// TwinCAT 3 PLC project TAC_Events
// Title: TAC_Events
// Company: Timberline Automation and Control Co.
// Author: Mit Patel
// ProjectVersion: 0.1.1.2
// Description: V0.1.1.0 - Initial V0.1.1.1 - Create RPC Sink V0.1.1.2 - Separate Buffer and Sink Interfaces
// ProgramVersion: 3.1.4026.19
// libraries:
//   Tc2_EtherCAT, * (Beckhoff Automation GmbH)
//   Tc2_Standard, * (Beckhoff Automation GmbH)
//   Tc2_System, * (Beckhoff Automation GmbH)
//   Tc2_Utilities, * (Beckhoff Automation GmbH)
//   Tc3_JsonXml, * (Beckhoff Automation GmbH)
// project tree:
//   ImportUtilities/ LogConfig.TcGVL
//   ImportUtilities/Logger/ E_LogSeverity.TcDUT, FB_LogErrorEdge.TcPOU, FB_LogInfoEdge.TcPOU, FB_LogOnEdge.TcPOU, FB_LogWarningEdge.TcPOU, F_LogDebug.TcPOU, F_LogError.TcPOU, F_Logger.TcPOU, F_LogInfo.TcPOU, F_LogWarning.TcPOU, I_ExternalLogger.TcIO
//   ImportUtilities/String/ F_Concat3.TcPOU, F_Concat4.TcPOU, F_Concat5.TcPOU, F_Concat6.TcPOU, F_Concat7.TcPOU, F_StringToTarg.TcPOU, F_TargToString.TcPOU, LongString.TcDUT
//   ImportUtilities/String/Large Concats/ F_ClearLarge.TcPOU, F_Concat3_Large.TcPOU, F_Concat4_Large.TcPOU, F_Concat5_Large.TcPOU, F_Concat6_Large.TcPOU, F_Concat7_Large.TcPOU, F_ConcatLarge.TcPOU
//   Library/EventLogger/EventBuffers/ T_JsonEventBuffer.TcPOU
//   Library/EventLogger/EventSinks/ T_RpcEventSink.TcPOU (not stored), FB_CsvFileEventSink.TcPOU (not stored)
//   Library/EventLogger/Interfaces/ I_EventSink.TcIO (not stored), I_EventBuffer.TcIO (not stored), I_EventLogger.TcIO (not stored), I_Logger.TcIO, I_EventSeverityHandler.TcIO (not stored), I_EventSinkHandler.TcIO
//   Library/Structs/ ST_EventMessageBuffer.TcDUT (not stored), ST_EventMessageBufferPool.TcDUT, ST_EventMessageParams.TcDUT, T_BufferString.TcDUT, T_MessageString.TcDUT (not stored)
//   Library/EventLogger/Bases/ T_InstanceNameBase.TcPOU (not stored)
//   Library/EventLogger/Functions/ F_GetLogSeverityFromTcEventSeverity.TcPOU (not stored)
//   Library/EventLogger/ T_EventLogger.TcPOU (not stored), T_Logger.TcPOU
//   Library/GVLs/ Events.TcGVL, EventsConfig.TcGVL (not stored)
//   Library/Time/ FB_UnixTimestamp.TcPOU, I_TimeProvider.TcIO (not stored)
//   Project Information/ F_GetCompany.TcPOU, F_GetTitle.TcPOU, F_GetVersion.TcPOU (not stored)
//   Version/ Global_Version.TcGVL
// real-time tasks:
//   TASK PlcTask: cycle T#10ms, priority 20, ADS port 350
//   TASK PlcTask1: cycle T#10ms, priority 21, ADS port 351

// ---- ImportUtilities/Logger/E_LogSeverity.TcDUT
{attribute 'qualified_only'}
TYPE
   E_LogSeverity :
   (
      Debug := 0,
      Info := ADSLOG_MSGTYPE_HINT,
      Warning := ADSLOG_MSGTYPE_WARN,
      Error := ADSLOG_MSGTYPE_ERROR,
      None := 1000
   ) DWORD;
END_TYPE

// ---- ImportUtilities/String/LongString.TcDUT
TYPE
   LongString : STRING(StringsParams.MAX_STRING_LENGTH);
END_TYPE // use StringsParams.MAX_STRING_LENGTH to adjust length

// ---- Library/Structs/ST_EventMessageBufferPool.TcDUT
{attribute 'pack_mode' := '0'}
TYPE ST_EventMessageBufferPool :
STRUCT
  bufferCount : UINT := EventsConfig.MAX_BUFFERS;
	currentDataBufferIndex : UINT := 0;
	dataBuffers : ARRAY [1..EventsConfig.MAX_BUFFERS] OF ST_EventMessageBuffer;
END_STRUCT
END_TYPE

// ---- Library/Structs/ST_EventMessageParams.TcDUT
TYPE ST_EventMessageParams :
STRUCT	
  Severity : TcEventSeverity;
  Message : T_MessageString;
  Source : T_MaxString;
END_STRUCT
END_TYPE

// ---- Library/Structs/T_BufferString.TcDUT
TYPE T_BufferString : STRING(EventsConfig.MAX_BUFFER_SIZE); END_TYPE

// ---- ImportUtilities/LogConfig.TcGVL
{attribute 'qualified_only'}
VAR_GLOBAL
   // set level to log. Lower log level includes higher levels i.e. info does warning and Error. 
   LogLevel : E_LogSeverity := E_LogSeverity.None; // Turn messages off by default
   ExternalLogger : I_ExternalLogger; // permit logging to something else
END_VAR

// ---- Library/GVLs/Events.TcGVL
{attribute 'qualified_only'}
VAR_GLOBAL CONSTANT
  {attribute 'hide'}
  {warning disable C0228}
  _eventLogger  : T_EventLogger;                      // Global instance of event logger which will log to all sinks.
  {warning restore C0228}

  EventLogger   : I_Logger := _eventLogger;           // Global accessor for logging events.
  EventSinks    : I_EventSinkHandler := _eventLogger; // Global accessor for adding/ resetting sinks.
END_VAR

// ---- Version/Global_Version.TcGVL
{attribute 'TcGenerated'}
{attribute 'no-analysis'}
{attribute 'linkalways'}
// This function has been automatically generated from the project information.
VAR_GLOBAL CONSTANT
	{attribute 'const_non_replaced'}
	stLibVersion_TAC_Events : ST_LibVersion := (iMajor := 0, iMinor := 1, iBuild := 1, iRevision := 2, nFlags := 0, sVersion := '0.1.1.2');
END_VAR

// ---- ImportUtilities/Logger/I_ExternalLogger.TcIO
INTERFACE I_ExternalLogger

METHOD AddToLog
VAR_IN_OUT
   Message : T_MaxString;
END_VAR
VAR_INPUT
   LogSeverity : E_LogSeverity;
END_VAR
END_METHOD

END_INTERFACE

// ---- Library/EventLogger/Interfaces/I_Logger.TcIO
// Interface for logging methods which can be called in user code.
INTERFACE I_Logger

METHOD LogCritical
VAR_INPUT
  message : T_MessageString; 
END_VAR
END_METHOD

METHOD LogError
VAR_INPUT
  message : T_MessageString; 
END_VAR
END_METHOD

METHOD LogInfo
VAR_INPUT
  message : T_MessageString; 
END_VAR
END_METHOD

METHOD LogVerbose
VAR_INPUT
  message : T_MessageString; 
END_VAR
END_METHOD

METHOD LogWarning
VAR_INPUT
  message : T_MessageString; 
END_VAR
END_METHOD

END_INTERFACE

// ---- Library/EventLogger/Interfaces/I_EventSinkHandler.TcIO
// Interface for handling sinks. Allows adding/ clearing sinks to be processed.
INTERFACE I_EventSinkHandler

// Adds a sink to the sink handler and returns TRUE if successful.
METHOD AddSink : BOOL
VAR_INPUT	
  sink : I_EventSink;
END_VAR
END_METHOD

// Clears all sinks currently being handled by the sink handler.
METHOD ClearSinks
END_METHOD

END_INTERFACE

// ---- ImportUtilities/Logger/FB_LogErrorEdge.TcPOU
FUNCTION_BLOCK FB_LogErrorEdge
VAR_INPUT
   Event : BOOL; // Event flag
   Message : T_MaxString; // Log message
   EventFallingEdge : BOOL := FALSE; // Defined which edge: FALSE = rising TRUE = falling, 
END_VAR
VAR_OUTPUT
   Q : BOOL;
END_VAR
VAR
   fbLogEdge : FB_LogOnEdge;
END_VAR

fbLogEdge(
   Event := Event,
   Message := Message,
   LogSeverity := E_LogSeverity.Error,
   EventFallingEdge := EventFallingEdge,
   Q => Q
);

END_FUNCTION_BLOCK

// ---- ImportUtilities/Logger/FB_LogOnEdge.TcPOU
FUNCTION_BLOCK FB_LogOnEdge
VAR_INPUT
   Event : BOOL; // look for edge here to log.
   Message : T_MaxString; // message
   LogSeverity : E_LogSeverity; // severity
   EventFallingEdge : BOOL := FALSE; // TRUE for falling edge, FALSE for rising edge.
END_VAR
VAR_OUTPUT
   Q : BOOL;
END_VAR
VAR
   rt : R_TRIG;
   ft : F_TRIG;
END_VAR
VAR_TEMP
   logNow : BOOL;
END_VAR

rt(CLK := Event);
ft(CLK := Event);

Q := SEL(EventFallingEdge, rt.Q, ft.Q);

IF Q THEN

   CASE LogSeverity OF

      E_LogSeverity.Info:
         F_LogInfo(Message);

      E_LogSeverity.Warning:
         F_LogWarning(Message);

      E_LogSeverity.Error:
         F_LogError(Message);
   ELSE

      F_LogError(
         CONCAT(
            'Error in FB_LogOnEdge, Logseverity incorrect. Log Message for event is : ',
            Message
         )
      );

   END_CASE

END_IF

END_FUNCTION_BLOCK

// ---- ImportUtilities/Logger/F_LogInfo.TcPOU
FUNCTION F_LogInfo : STRING;
VAR_INPUT
   Message : T_MaxString;
END_VAR

F_LogInfo := F_Logger(ADSLOG_MSGTYPE_HINT, Message);

END_FUNCTION

// ---- ImportUtilities/Logger/F_Logger.TcPOU
FUNCTION F_Logger : STRING;
VAR_INPUT
   LogSeverity : E_LogSeverity;
   Message : T_MaxString;
END_VAR

IF (LogSeverity < E_LogSeverity.None)
   AND_THEN (LogSeverity >= LogConfig.LogLevel) THEN

   ADSLOGSTR(LogSeverity OR ADSLOG_MSGTYPE_LOG, Message, '');
   F_Logger := Message;

   IF LogConfig.ExternalLogger <> 0 THEN
      LogConfig.ExternalLogger.AddToLog(Message, LogSeverity);
   END_IF

END_IF

END_FUNCTION

// ---- ImportUtilities/Logger/F_LogWarning.TcPOU
FUNCTION F_LogWarning : STRING;
VAR_INPUT
   Message : T_MaxString;
END_VAR

F_LogWarning := F_Logger(ADSLOG_MSGTYPE_WARN, Message);

END_FUNCTION

// ---- ImportUtilities/Logger/F_LogError.TcPOU
FUNCTION F_LogError : STRING;
VAR_INPUT
   Message : T_MaxString;
END_VAR

F_LogError := F_Logger(ADSLOG_MSGTYPE_ERROR, Message);

END_FUNCTION

// ---- ImportUtilities/Logger/FB_LogInfoEdge.TcPOU
FUNCTION_BLOCK FB_LogInfoEdge
VAR_INPUT
   Event : BOOL; // Event flag
   Message : T_MaxString; // Log message
   EventFallingEdge : BOOL := FALSE; // Defined which edge: FALSE = rising TRUE = falling, 
END_VAR
VAR_OUTPUT
   Q : BOOL;
END_VAR
VAR
   fbLogEdge : FB_LogOnEdge;
END_VAR

fbLogEdge(
   Event := Event,
   Message := Message,
   LogSeverity := E_LogSeverity.Info,
   EventFallingEdge := EventFallingEdge,
   Q => Q
);

END_FUNCTION_BLOCK

// ---- ImportUtilities/Logger/FB_LogWarningEdge.TcPOU
FUNCTION_BLOCK FB_LogWarningEdge
VAR_INPUT
   Event : BOOL; // Event flag
   Message : T_MaxString; // Log message
   EventFallingEdge : BOOL := FALSE; // Defined which edge: FALSE = rising TRUE = falling, 
END_VAR
VAR_OUTPUT
   Q : BOOL;
END_VAR
VAR
   fbLogEdge : FB_LogOnEdge;
END_VAR

fbLogEdge(
   Event := Event,
   Message := Message,
   LogSeverity := E_LogSeverity.Warning,
   EventFallingEdge := EventFallingEdge,
   Q => Q
);

END_FUNCTION_BLOCK

// ---- ImportUtilities/Logger/F_LogDebug.TcPOU
FUNCTION F_LogDebug : STRING;
VAR_INPUT
   Message : T_MaxString;
END_VAR

F_LogDebug :=
   F_Logger(
      E_LogSeverity.Debug,
      CONCAT('DEBUG ', Message)
   );

END_FUNCTION

// ---- ImportUtilities/String/F_Concat3.TcPOU
FUNCTION F_Concat3 : T_MaxString
VAR_INPUT
   StringOne : STRING;
   StringTwo : STRING;
   StringThree : STRING;
END_VAR
VAR
   response : T_MaxString;
END_VAR

response := CONCAT(StringOne, StringTwo);
response := CONCAT(response, StringThree);
F_Concat3 := response;

END_FUNCTION

// ---- ImportUtilities/String/F_Concat4.TcPOU
FUNCTION F_Concat4 : T_MaxString
VAR_INPUT
   sOne : STRING;
   sTwo : STRING;
   sThree : STRING;
   sFour : STRING;
END_VAR

F_Concat4 := CONCAT(
   sOne,
   F_Concat3(sTwo, sThree, sFour)
);

END_FUNCTION

// ---- ImportUtilities/String/F_Concat5.TcPOU
FUNCTION F_Concat5 : T_MaxString
VAR_INPUT
   sOne : STRING;
   sTwo : STRING;
   sThree : STRING;
   sFour : STRING;
   sFive : STRING;
END_VAR

F_Concat5 := CONCAT(
   sOne,
   F_Concat4(sTwo, sThree, sFour, sFive)
);

END_FUNCTION

// ---- ImportUtilities/String/F_Concat6.TcPOU
FUNCTION F_Concat6 : T_MaxString
VAR_INPUT
   sOne : STRING;
   sTwo : STRING;
   sThree : STRING;
   sFour : STRING;
   sFive : STRING;
   sSix : STRING;
END_VAR

F_Concat6 := CONCAT(
   sOne,
   F_Concat5(sTwo, sThree, sFour, sFive, sSix)
);

END_FUNCTION

// ---- ImportUtilities/String/F_Concat7.TcPOU
FUNCTION F_Concat7 : T_MaxString
VAR_INPUT
   sOne : STRING;
   sTwo : STRING;
   sThree : STRING;
   sFour : STRING;
   sFive : STRING;
   sSix : STRING;
   sSeven : STRING;
END_VAR

F_Concat7 := CONCAT(
   sOne,
   F_Concat6(
      sTwo,
      sThree,
      sFour,
      sFive,
      sSix,
      sSeven
   )
);

END_FUNCTION

// ---- ImportUtilities/String/F_StringToTarg.TcPOU
FUNCTION F_StringToTarg
VAR_INPUT
   StringToConvert : T_MaxString;
END_VAR
VAR_IN_OUT
   Targ : T_ARG;
END_VAR
VAR
   b : POINTER TO BOOL;
   b8 : POINTER TO BYTE;
   w : POINTER TO WORD;
   dw : POINTER TO DWORD;
   usi : POINTER TO USINT;
   si : POINTER TO SINT;
   ui : POINTER TO UINT;
   i : POINTER TO INT;
   udi : POINTER TO UDINT;
   di : POINTER TO DINT;
   str : POINTER TO STRING;
   re : POINTER TO REAL;
   lr : POINTER TO LREAL;
END_VAR

CASE Targ.eType OF

   E_ArgType.ARGTYPE_BOOL:
      b := Targ.pData;
      b^ := TO_BOOL(StringToConvert);

   E_ArgType.ARGTYPE_BYTE:
      b8 := Targ.pData;
      b8^ := TO_BYTE(StringToConvert);

   E_ArgType.ARGTYPE_WORD:
      w := Targ.pData;
      w^ := TO_WORD(StringToConvert);

   E_ArgType.ARGTYPE_DWORD:
      dw := Targ.pData;
      dw^ := TO_DWORD(StringToConvert);

   E_ArgType.ARGTYPE_USINT:
      usi := Targ.pData;
      usi^ := TO_USINT(StringToConvert);

   E_ArgType.ARGTYPE_SINT:
      si := Targ.pData;
      si^ := TO_SINT(StringToConvert);

   E_ArgType.ARGTYPE_UINT:
      ui := Targ.pData;
      ui^ := TO_UINT(StringToConvert);

   E_ArgType.ARGTYPE_INT:
      i := Targ.pData;
      i^ := TO_INT(StringToConvert);

   E_ArgType.ARGTYPE_UDINT:
      udi := Targ.pData;
      udi^ := TO_UDINT(StringToConvert);

   E_ArgType.ARGTYPE_DINT:
      di := Targ.pData;
      di^ := TO_DINT(StringToConvert);

   E_ArgType.ARGTYPE_STRING:
      str := Targ.pData;
      str^ := TO_STRING(StringToConvert);

   E_ArgType.ARGTYPE_REAL:
      re := Targ.pData;
      re^ := TO_REAL(StringToConvert);

   E_ArgType.ARGTYPE_LREAL:
      lr := Targ.pData;
      lr^ := TO_LREAL(StringToConvert);

ELSE
   F_LogWarning(
      CONCAT(
         'Unsupported type in Targ for string conversion: ',
         TO_STRING(Targ.eType)
      )
   );
END_CASE

END_FUNCTION

// ---- ImportUtilities/String/F_TargToString.TcPOU
FUNCTION F_TargToString : T_MaxString
VAR_INPUT
   Targ : T_ARG;
END_VAR
VAR
   b : POINTER TO BOOL;
   b8 : POINTER TO BYTE;
   w : POINTER TO WORD;
   dw : POINTER TO DWORD;
   usi : POINTER TO USINT;
   si : POINTER TO SINT;
   ui : POINTER TO UINT;
   i : POINTER TO INT;
   udi : POINTER TO UDINT;
   di : POINTER TO DINT;
   str : POINTER TO STRING;
   re : POINTER TO REAL;
   lr : POINTER TO LREAL;
END_VAR

CASE Targ.eType OF

   E_ArgType.ARGTYPE_BOOL:
      b := Targ.pData;
      F_TargToString := TO_STRING(b^);

   E_ArgType.ARGTYPE_BYTE:
      b8 := Targ.pData;
      F_TargToString := TO_STRING(b8^);

   E_ArgType.ARGTYPE_WORD:
      w := Targ.pData;
      F_TargToString := TO_STRING(w^);

   E_ArgType.ARGTYPE_DWORD:
      dw := Targ.pData;
      F_TargToString := TO_STRING(dw^);

   E_ArgType.ARGTYPE_USINT:
      usi := Targ.pData;
      F_TargToString := TO_STRING(usi^);

   E_ArgType.ARGTYPE_SINT:
      si := Targ.pData;
      F_TargToString := TO_STRING(si^);

   E_ArgType.ARGTYPE_UINT:
      ui := Targ.pData;
      F_TargToString := TO_STRING(ui^);

   E_ArgType.ARGTYPE_INT:
      i := Targ.pData;
      F_TargToString := TO_STRING(i^);

   E_ArgType.ARGTYPE_UDINT:
      udi := Targ.pData;
      F_TargToString := TO_STRING(udi^);

   E_ArgType.ARGTYPE_DINT:
      di := Targ.pData;
      F_TargToString := TO_STRING(di^);

   E_ArgType.ARGTYPE_STRING:
      str := Targ.pData;
      F_TargToString := TO_STRING(str^);

   E_ArgType.ARGTYPE_REAL:
      re := Targ.pData;
      F_TargToString := TO_STRING(re^);

   E_ArgType.ARGTYPE_LREAL:
      lr := Targ.pData;
      F_TargToString := TO_STRING(lr^);

ELSE
   F_LogWarning(
      CONCAT(
         'Unsupported type in Targ for string conversion: ',
         TO_STRING(Targ.eType)
      )
   );
END_CASE

END_FUNCTION

// ---- ImportUtilities/String/Large Concats/F_ClearLarge.TcPOU
FUNCTION F_ClearLarge
VAR_IN_OUT CONSTANT
   stringToClear : LongString;
END_VAR

MEMSET(ADR(stringToClear), 16#0, sizeof(stringToClear));

END_FUNCTION

// ---- ImportUtilities/String/Large Concats/F_Concat3_Large.TcPOU
FUNCTION F_Concat3_Large : LongString;
VAR_IN_OUT CONSTANT
   StringOne : LongString;
   StringTwo : LongString;
   StringThree : LongString;
END_VAR
VAR
   str : LongString;
END_VAR

str := F_ConcatLarge(StringTwo, StringThree);

F_Concat3_Large :=
   F_ConcatLarge(
      StringOne,
      str
   );

END_FUNCTION

// ---- ImportUtilities/String/Large Concats/F_ConcatLarge.TcPOU
FUNCTION F_ConcatLarge : LongString
VAR_IN_OUT CONSTANT
   StringOne : LongString;
   StringTwo : LongString;
END_VAR
VAR
   i, sizeToCpy, teminatingCharPos, maxLen : DINT;
   response : LongString;
END_VAR

maxLen := TO_DINT(StringsParams.MAX_STRING_LENGTH) - 1; // - 1 allows for terminating character in last position.

IF LEN(stringOne) + LEN(StringTwo) > maxLen THEN
   sizeToCpy := maxLen - LEN(StringTwo); //need room for the terminating character
   teminatingCharPos := maxLen; // this is the index position for utf-8 string as byte array

ELSE
   sizeToCpy := LEN(StringOne);
   teminatingCharPos := LEN(StringOne) + LEN(StringTwo);

END_IF

// copy strings into response
MEMCPY(ADR(response), ADR(StringOne), TO_UDINT(sizeToCpy));
MEMCPY(ADR(response[sizeToCpy]), ADR(StringTwo), TO_UDINT(LEN(StringTwo)));

response[teminatingCharPos] := 16#0; // string terminating character
F_ConcatLarge := response;

END_FUNCTION

// ---- ImportUtilities/String/Large Concats/F_Concat4_Large.TcPOU
FUNCTION F_Concat4_Large : LongString
VAR_IN_OUT CONSTANT
   sOne : LongString;
   sTwo : LongString;
   sThree : LongString;
   sFour : LongString;
END_VAR
VAR
   str : LongString;
END_VAR

str := F_Concat3_Large(sTwo, sThree, sFour);

F_Concat4_Large :=
   F_ConcatLarge(
      sOne,
      str
   );

END_FUNCTION

// ---- ImportUtilities/String/Large Concats/F_Concat5_Large.TcPOU
FUNCTION F_Concat5_Large : LongString
VAR_IN_OUT CONSTANT
   sOne : LongString;
   sTwo : LongString;
   sThree : LongString;
   sFour : LongString;
   sFive : LongString;
END_VAR
VAR
   str : LongString;
END_VAR

str := F_Concat4_Large(sTwo, sThree, sFour, sFive);
F_Concat5_Large :=
   F_ConcatLarge(
      sOne,
      str
   );

END_FUNCTION

// ---- ImportUtilities/String/Large Concats/F_Concat6_Large.TcPOU
FUNCTION F_Concat6_Large : LongString
VAR_IN_OUT CONSTANT
   sOne : LongString;
   sTwo : LongString;
   sThree : LongString;
   sFour : LongString;
   sFive : LongString;
   sSix : LongString;
END_VAR
VAR
   str : LongString;
END_VAR

str := F_Concat5_Large(sTwo, sThree, sFour, sFive, sSix);
F_Concat6_Large :=
   F_ConcatLarge(
      sOne,
      str
   );

END_FUNCTION

// ---- ImportUtilities/String/Large Concats/F_Concat7_Large.TcPOU
FUNCTION F_Concat7_Large : LongString
VAR_IN_OUT CONSTANT
   sOne : LongString;
   sTwo : LongString;
   sThree : LongString;
   sFour : LongString;
   sFive : LongString;
   sSix : LongString;
   sSeven : LongString;
END_VAR
VAR
   str : LongString;
END_VAR

str := F_Concat6_Large(
   sTwo,
   sThree,
   sFour,
   sFive,
   sSix,
   sSeven
);

F_Concat7_Large :=
   F_ConcatLarge(
      sOne,
      str
   );

END_FUNCTION

// ---- Library/EventLogger/EventBuffers/T_JsonEventBuffer.TcPOU
// Event sink which buffers log messages/ events ready for polling via RPC calls to 'GetEvents'; a method of the I_EventSink interface. 
FUNCTION_BLOCK PUBLIC T_JsonEventBuffer EXTENDS T_InstanceNameBase IMPLEMENTS I_EventBuffer
VAR
  isInitialised : BOOL := FALSE;
  
  bufferPool : ST_EventMessageBufferPool;
  jWriters : ARRAY [1..EventsConfig.MAX_BUFFERS] OF FB_JsonSaxWriter;

  _timeProvider : I_TimeProvider := NULL;
  eventId : ULINT := 0;
END_VAR

VAR CONSTANT
  NULL : UDINT := 0;
END_VAR

// Adds an event to the buffer for later processing.
METHOD PUBLIC AddEvent
VAR_INPUT
  eventMessageParams : ST_EventMessageParams;
END_VAR

VAR
  totalSize, messageSize : UDINT := 0;
  buffer : REFERENCE TO ST_EventMessageBuffer := 0;
END_VAR

VAR_INST
  jWriterLocal : FB_JsonSaxWriter; // For calculating message size.
END_VAR

VAR CONSTANT
  END_JSON_ARRAY_SIZE : UINT := 3; // End array, end object and null terminator.
END_VAR
IF NOT isInitialised THEN
  F_LogWarning(CONCAT(InstanceName, ': Unable to AddEvent. Sink is uninitialised.'));
  RETURN;
END_IF

jWriterLocal.ResetDocument();
messageSize := ConvertToJson(eventMessageParams, jWriter := jWriterLocal);

IF bufferPool.currentDataBufferIndex = 0 OR bufferPool.currentDataBufferIndex > EventsConfig.MAX_BUFFERS THEN // Try to find an empty buffer.
	bufferPool.currentDataBufferIndex := FindAvailableBuffer();
  ResetBuffer(bufferPool.currentDataBufferIndex);
END_IF

IF bufferPool.currentDataBufferIndex > 0 AND bufferPool.currentDataBufferIndex <= EventsConfig.MAX_BUFFERS THEN 
  buffer REF= bufferPool.dataBuffers[bufferPool.currentDataBufferIndex];

  IF buffer.dataSize + messageSize > (EventsConfig.MAX_BUFFER_SIZE - END_JSON_ARRAY_SIZE) THEN  // Will adding this event cause the buffer to overflow?
    EndJson(bufferPool.currentDataBufferIndex);
    buffer.availableForWriting := FALSE; // Available for reading/ sending

	  bufferPool.currentDataBufferIndex := FindAvailableBuffer(); // Next buffer for writing. Will return 0 if no available buffers.
    ResetBuffer(bufferPool.currentDataBufferIndex);
  END_IF
END_IF

IF bufferPool.currentDataBufferIndex > 0 AND bufferPool.currentDataBufferIndex <= EventsConfig.MAX_BUFFERS THEN // Check bounds again due to buffer index change above.
  buffer REF= bufferPool.dataBuffers[bufferPool.currentDataBufferIndex]; // Buffer index has changed so update the internal ref.
  IF buffer.availableForWriting THEN
    ConvertToJson(eventMessageParams, jWriter := jWriters[bufferPool.currentDataBufferIndex]);
    totalSize := jWriters[bufferPool.currentDataBufferIndex].GetDocumentLength();                 
    buffer.dataSize := totalSize;
    buffer.count := buffer.count + 1;
    eventId := eventId + 1;
  END_IF
END_IF
END_METHOD

// Converts the input eventMessageParams to JSON (without string copying).
METHOD PRIVATE ConvertToJson
VAR_INPUT
  eventMessageParams : ST_EventMessageParams;
END_VAR

VAR_OUTPUT
  docSize : UDINT;
END_VAR

VAR_IN_OUT
  jWriter : FB_JsonSaxWriter;
END_VAR

VAR
  timestampMs : ULINT;
  severity : T_MaxString;
END_VAR
IF NOT isInitialised THEN
  F_LogWarning(CONCAT(InstanceName, ': Unable to ConvertToJson. Sink is uninitialised.'));
  RETURN;
END_IF

IF _timeProvider = NULL THEN
  F_LogWarning(CONCAT(InstanceName, ': Unable to ConvertToJson. _timeProvider is uninitialised.'));
  RETURN;
END_IF

timestampMs := _timeProvider.TimestampMs;
severity := TO_STRING(eventMessageParams.Severity);

jWriter.StartObject();

  jWriter.AddKey('EventId');
  jWriter.AddUlint(eventId);

  jWriter.AddKeyString('Severity', severity);
  jWriter.AddKey('FileTime'); // Add unix timestamp
  jWriter.AddUlint(timestampMs);
  jWriter.AddKeyString('SourceName', eventMessageParams.Source); 
  jWriter.AddKeyString('MessageBody', eventMessageParams.Message);
  
jWriter.EndObject();

docSize := jWriter.GetDocumentLength();
END_METHOD

// Copies data in the JSON writer and returns the total length of bytes copied.
METHOD PRIVATE CopyJson : UDINT
VAR_INPUT
  iBuffer : UINT := 0;
  resultString : REFERENCE TO T_BufferString;
END_VAR

VAR
  totalSize : UDINT := 0;
END_VAR

VAR CONSTANT
  RESULT_STRING_SIZE : UDINT := SIZEOF(resultString);
END_VAR
IF NOT isInitialised THEN
  F_LogWarning(CONCAT(InstanceName, ': Unable to CopyJson. Sink is uninitialised.'));
  RETURN;
END_IF

IF iBuffer = 0 OR iBuffer > EventsConfig.MAX_BUFFERS THEN
	RETURN;
END_IF

MEMSET(ADR(resultString), 0, RESULT_STRING_SIZE); // Copy doc should overwrite resultString including null termination characters. 

totalSize := jWriters[iBuffer].CopyDocument
             (
               PDoc := resultString, 
               nDoc := RESULT_STRING_SIZE
             );
             
bufferPool.dataBuffers[iBuffer].dataSize := totalSize;
CopyJson := totalSize;
END_METHOD

// Ends the JSON string, ready for the JSON string to be copied.
METHOD PRIVATE EndJson
VAR_INPUT
  iBuffer : UINT := 0;
END_VAR
IF NOT isInitialised THEN
  F_LogWarning(CONCAT(InstanceName, ': Unable to EndJson. Sink is uninitialised.'));
  RETURN;
END_IF

IF iBuffer = 0 OR iBuffer > EventsConfig.MAX_BUFFERS THEN
	RETURN;
END_IF

jWriters[iBuffer].EndArray();
jWriters[iBuffer].EndObject();
END_METHOD

// Finds the first available buffer, if unable to find one and CYCLE_BUFFERS is set to TRUE, then will search for the first oldest buffer based on its timestamp.
// With CYCLE_BUFFERS set to FALSE, events will be dropped.
// Returns the buffer index from the pool, 0 (invalid) if a buffer is not found.
METHOD PRIVATE FindAvailableBuffer : UINT
VAR
  iBuffer : UINT := 0;
  iAvailable : UINT := 0;
  iOldest : UINT := 0;
END_VAR
IF NOT isInitialised THEN
  F_LogWarning(CONCAT(InstanceName, ': Unable to FindAvailableBuffer. Sink is uninitialised.'));
  RETURN;
END_IF

iAvailable := 0;

FOR iBuffer := 1 TO EventsConfig.MAX_BUFFERS DO 
  IF bufferPool.dataBuffers[iBuffer].availableForWriting THEN
    iAvailable := iBuffer;
    EXIT;
	END_IF
END_FOR

IF EventsConfig.CYCLE_BUFFERS THEN
  // All buffers are full
  IF iAvailable = 0 THEN
    iOldest := FindOldestBuffer(FALSE);
    IF iOldest > 0 AND iOldest <= EventsConfig.MAX_BUFFERS THEN
      iAvailable := iOldest;
    END_IF
  END_IF
END_IF

FindAvailableBuffer := iAvailable;
END_METHOD

// Finds the oldest buffer in the pool and returns its buffer index. Will return 0 if unable to find an old buffer.
// If checkHasItems is set to TRUE, then will only search for buffers with items, otherwise all buffers in the pool are considered.
METHOD PRIVATE FindOldestBuffer : UINT
VAR_INPUT
  checkHasItems : BOOL := FALSE;
END_VAR

VAR
  iBuffer : UINT := 0;
  iOldest : UINT := 0;
  timeOldest : ULINT;
END_VAR
IF NOT isInitialised THEN
  F_LogWarning(CONCAT(InstanceName, ': Unable to FindOldestBuffer. Sink is uninitialised.'));
  RETURN;
END_IF

IF _timeProvider = NULL THEN
  F_LogWarning(CONCAT(InstanceName, ': Unable to FindOldestBuffer. _timeProvider is uninitialised.'));
  RETURN;
END_IF

timeOldest := _timeProvider.TimestampMs;
FOR iBuffer := 1 TO EventsConfig.MAX_BUFFERS DO
  IF bufferPool.dataBuffers[iBuffer].timestampMs < timeOldest THEN
    IF NOT checkHasItems OR_ELSE bufferPool.dataBuffers[iBuffer].count > 0 THEN
      timeOldest := bufferPool.dataBuffers[iBuffer].timestampMs;
      iOldest := iBuffer;
    END_IF
  END_IF
END_FOR
    
FindOldestBuffer := iOldest;
END_METHOD

// Gets events currently stored in the buffer and copies them to the resultString, returning the total length of bytes copied.
METHOD PUBLIC GetEvents : UDINT
VAR_INPUT
  resultString : REFERENCE TO T_BufferString;
END_VAR

VAR
  iBuffer : UINT := 0;
  totalSize : UDINT := 0;
END_VAR

VAR CONSTANT
  // Note that the size returned from any 
  // json writer's GetDocumentLength method 
  // includes the null terminator, which we want to remove.
  // This is due to the JSON parsers in .NET or Influx's Telegraf, etc
  // not being able to understand the null terminator and throwing errors,
  // e.g. stating that there are additional characters at the end of the JSON payload.
  REMOVE_NULL_TERMINATOR : UDINT := 1;
END_VAR
IF NOT isInitialised THEN
  F_LogWarning(CONCAT(InstanceName, ': Unable to GetEvents. Sink is uninitialised.'));
  RETURN;
END_IF

iBuffer := FindOldestBuffer(TRUE);
IF iBuffer > 0 AND iBuffer <= EventsConfig.MAX_BUFFERS THEN
  IF NOT bufferPool.dataBuffers[iBuffer].availableForWriting THEN
    IF bufferPool.dataBuffers[iBuffer].count > 0 THEN
      totalSize := CopyJson(iBuffer, resultString);
      ResetBuffer(iBuffer);
    END_IF
  ELSE // Current buffer
    IF bufferPool.dataBuffers[iBuffer].count > 0 THEN
      bufferPool.dataBuffers[iBuffer].availableForWriting := FALSE; // Available for reading/ sending
      EndJson(iBuffer);
      totalSize := CopyJson(iBuffer, resultString);
      ResetBuffer(iBuffer);
      bufferPool.currentDataBufferIndex := FindAvailableBuffer(); // Next buffer for writing. Will return 0 if no available buffers.
      ResetBuffer(bufferPool.currentDataBufferIndex);
    END_IF
  END_IF
END_IF

GetEvents := totalSize - REMOVE_NULL_TERMINATOR;
END_METHOD

// Initialises the buffer including an I_TimeProvider for timestamping buffers and events.
METHOD PUBLIC Initialise
VAR_INPUT
	timeProvider : I_TimeProvider;
END_VAR

VAR
  iBuffer : UINT := 0;
END_VAR
_timeProvider := timeProvider;

IF _timeProvider = NULL THEN
  F_LogWarning(CONCAT(InstanceName, ': Unable to Initialise. _timeProvider is uninitialised.'));
  RETURN;
END_IF

isInitialised := TRUE;

FOR iBuffer := 1 TO EventsConfig.MAX_BUFFERS DO 
  ResetBuffer(iBuffer);
END_FOR
END_METHOD

// Resets a buffer based on the input buffer index and starts the buffer ready for new events to be added.
METHOD PRIVATE ResetBuffer
VAR_INPUT
  iBuffer : UINT := 0;
END_VAR
IF NOT isInitialised THEN
  F_LogWarning(CONCAT(InstanceName, ': Unable to ResetBuffer. Sink is uninitialised.'));
  RETURN;
END_IF

IF _timeProvider = NULL THEN
  F_LogWarning(CONCAT(InstanceName, ': Unable to ResetBuffer. _timeProvider is uninitialised.'));
  RETURN;
END_IF

IF iBuffer > 0 AND iBuffer <= EventsConfig.MAX_BUFFERS THEN
  StartJson(iBuffer);
  
  bufferPool.dataBuffers[iBuffer].bufferIndex := iBuffer;
  bufferPool.dataBuffers[iBuffer].availableForWriting := TRUE;
  bufferPool.dataBuffers[iBuffer].count := 0;
  bufferPool.dataBuffers[iBuffer].bufferSize := EventsConfig.MAX_BUFFER_SIZE;
  bufferPool.dataBuffers[iBuffer].dataSize := 0;
  
  bufferPool.dataBuffers[iBuffer].timestampMs := _timeProvider.TimestampMs;
END_IF
END_METHOD

// Starts the JSON string, for additional JSON objects can be appended.
METHOD PRIVATE StartJson
VAR_INPUT
  iBuffer : UINT := 0;
END_VAR
IF NOT isInitialised THEN
  F_LogWarning(CONCAT(InstanceName, ': Unable to StartJson. Sink is uninitialised.'));
  RETURN;
END_IF

IF iBuffer = 0 OR iBuffer > EventsConfig.MAX_BUFFERS THEN
	RETURN;
END_IF

jWriters[iBuffer].ResetDocument();  
jWriters[iBuffer].StartObject();
jWriters[iBuffer].AddKey('Logs');
jWriters[iBuffer].StartArray();
END_METHOD

END_FUNCTION_BLOCK

// ---- Library/EventLogger/T_Logger.TcPOU
// Logger for allowing events of any level to be raised in addition to being able to set/clear a local severity for specific logs.
FUNCTION_BLOCK PUBLIC T_Logger EXTENDS T_InstanceNameBase IMPLEMENTS I_EventLogger, I_Logger, I_EventSeverityHandler
VAR CONSTANT
  NULL : UDINT := 0;
END_VAR

// Clear the currently set local severity level.
METHOD PUBLIC ClearLocalSeverity
Events._eventLogger.ClearLocalSeverity();
END_METHOD

{attribute 'hide'}
METHOD FB_init : BOOL
VAR_INPUT
	bInitRetains : BOOL; // if TRUE, the retain variables are initialized (warm start / cold start)
	bInCopyCode : BOOL;  // if TRUE, the instance afterwards gets moved into the copy code (online change)
END_VAR
// Ensure Intecre_Utilities log level is set to Debug so all logs are processed. 
// Log filtering is handled via Events.GLOBAL_LOG_SEVERITY and I_Logger -> I_EventSeverityHandler for setting local severity.
// See events tester.
//Intecre_Utilities.LogConfig.LogLevel := E_LogSeverity.Debug; 

// Set the minimum global logging severity to filter all events.
SetGlobalSeverity(TcEventSeverity.Verbose);
END_METHOD

// Get global severity level.
METHOD GetGlobalSeverity : TcEventSeverity
GetGlobalSeverity := Events._eventLogger.GetGlobalSeverity();
END_METHOD

// Get local severity level.
METHOD GetLocalSeverity : TcEventSeverity
GetLocalSeverity := Events._eventLogger.GetLocalSeverity();
END_METHOD

METHOD PUBLIC LogCritical
VAR_INPUT
	message	: T_MessageString;
END_VAR

VAR
  localInstanceName : T_MaxString;
END_VAR
localInstanceName := InstanceName;
LogEvent(message := message, sourceInstanceName := localInstanceName, severity := TcEventSeverity.Critical);;
END_METHOD

METHOD PUBLIC LogError
VAR_INPUT
	message	: T_MessageString;
END_VAR

VAR
  localInstanceName : T_MaxString;
END_VAR
localInstanceName := InstanceName;
LogEvent(message := message, sourceInstanceName := localInstanceName, severity := TcEventSeverity.Error);
END_METHOD

METHOD INTERNAL LogEvent
VAR_IN_OUT CONSTANT
  message : T_MessageString; 
  sourceInstanceName : T_MaxString;
END_VAR

VAR_INPUT
  severity : TcEventSeverity;
END_VAR
IF Events.EventLogger = NULL THEN
  F_LogWarning(CONCAT(InstanceName, ': Unable to LogEvent. Events.EventLogger is null/ uninitialised.'));
  RETURN;
END_IF

IF NOT ShouldLogEvent(severity) THEN
  RETURN;
END_IF

Events._eventLogger.LogEvent(
    message:= message, 
    sourceInstanceName:= sourceInstanceName, 
    severity:= severity
  );
END_METHOD

METHOD PUBLIC LogInfo
VAR_INPUT
	message	: T_MessageString;
END_VAR

VAR
  localInstanceName : T_MaxString;
END_VAR
localInstanceName := InstanceName;
LogEvent(message := message, sourceInstanceName := localInstanceName, severity := TcEventSeverity.Info);
END_METHOD

METHOD PUBLIC LogVerbose
VAR_INPUT
	message	: T_MessageString;
END_VAR

VAR
  localInstanceName : T_MaxString;
END_VAR
localInstanceName := InstanceName;
LogEvent(message := message, sourceInstanceName := localInstanceName, severity := TcEventSeverity.Verbose);
END_METHOD

METHOD PUBLIC LogWarning
VAR_INPUT
	message	: T_MessageString;
END_VAR

VAR
  localInstanceName : T_MaxString;
END_VAR
localInstanceName := InstanceName;
LogEvent(message := message, sourceInstanceName := localInstanceName, severity := TcEventSeverity.Warning);
END_METHOD

// Set a global severity level to filter logged events.
METHOD PUBLIC SetGlobalSeverity
VAR_INPUT
	severity	: TcEventSeverity;
END_VAR
Events._eventLogger.SetGlobalSeverity(severity);
END_METHOD

// Set a local severity level to filter logged events. Ensure clear is called once local logging is complete.
METHOD PUBLIC SetLocalSeverity
VAR_INPUT
	severity	: TcEventSeverity;
END_VAR
Events._eventLogger.SetLocalSeverity(severity);
END_METHOD

METHOD INTERNAL ShouldLogEvent : BOOL
VAR_INPUT
  severity : TcEventSeverity;
END_VAR
ShouldLogEvent := TRUE;
END_METHOD

END_FUNCTION_BLOCK

// ---- Library/Time/FB_UnixTimestamp.TcPOU
// Timestamp provider for calculating Unix time. Required to be called in a cyclic manner.
FUNCTION_BLOCK PUBLIC FB_UnixTimestamp IMPLEMENTS I_TimeProvider
VAR_OUTPUT
	milliseconds : ULINT;
	cpuMicroSeconds : ULINT;
	systemMicroSeconds : ULINT;
	dcToTimeZoneMicroSeconds : ULINT;
END_VAR

VAR
	localSystemTime : FB_LocalSystemTime := (bEnable := TRUE, dwCycle := 1);
	getTimeZoneInformation : FB_GetTimeZoneInformation;
	timeZoneInformation : ST_TimeZoneInformation;
	specificLocalTimeToFileTime, specificDcToFileTime : FB_TzSpecificLocalTimeToFileTime;
	fileTime, dcFileTime, dcToFileTime : T_FILETIME;
	onZerothSecondLastCycle : BOOL;
	tDcTime : T_DCTIME64;

	cpuHighTime, systemHighTime : UDINT;
	cpuLowTime, systemLowTime : UDINT;
	getSystemTime : GETSYSTEMTIME;
	getCPUCounter : GETCPUCOUNTER;
	diffBetweenSystemAndDc, prevDiff : ULINT;
  _timestampMs : ULINT;
END_VAR

// Get local system time
tDcTime := F_GetCurDcTaskTime64();
localSystemTime();
getCPUCounter( cpuCntHiDW => cpuHighTime, cpuCntLoDW => cpuLowTime );
getSystemTime( timeHiDW => systemHighTime, timeLoDW => systemLowTime );

// On the zeroth second of each minutesync timezone information
IF (timeZoneInformation.standardName = '' OR (localSystemTime.systemTime.wSecond = 0 AND NOT onZerothSecondLastCycle)) THEN
	getTimeZoneInformation( sNetID := '', bExecute := TRUE, tzInfo => timeZoneInformation );
END_IF;

// Convert local system time to unix timestamps
specificLocalTimeToFileTime(
		in := Tc2_Utilities.SYSTEMTIME_TO_FILETIME( localSystemTime.systemTime ),
		tzInfo := timeZoneInformation,
		out => fileTime
	);

_timestampMs := milliseconds := (SHL( DWORD_TO_ULINT( fileTime.dwHighDateTime ), 32 ) + DWORD_TO_ULINT( fileTime.dwLowDateTime )) / 10000 - 11644473600000;

onZerothSecondLastCycle := localSystemTime.systemTime.wSecond = 0;

specificDcToFileTime( in := DCTIME64_TO_FILETIME( tDcTime ), tzInfo := timeZoneInformation, out => dcFileTime );
dcToTimeZoneMicroSeconds :=
	(SHL( DWORD_TO_ULINT( dcFileTime.dwHighDateTime ), 32 ) + DWORD_TO_ULINT( dcFileTime.dwLowDateTime )) / 10 - 11644473600000000;

cpuMicroSeconds := (SHL( DWORD_TO_ULINT( cpuHighTime ), 32 ) + DWORD_TO_ULINT( cpuLowTime )) / 10 - 11644473600000000;
systemMicroSeconds := (SHL( DWORD_TO_ULINT( systemHighTime ), 32 ) + DWORD_TO_ULINT( systemLowTime )) / 10 - 11644473600000000;

//diffBetweenSystemAndDc := dcToTimeZoneMilliSeconds - localSysTimeMlSec;

PROPERTY TimestampMs : ULINT
GET
TimestampMs := milliseconds;
END_GET
END_PROPERTY

END_FUNCTION_BLOCK

// ---- Project Information/F_GetCompany.TcPOU
// This function has been automatically generated from the project information.
{attribute 'signature_flag' := '1073741824'}
{attribute 'TcGenerated'}
{attribute 'no-analysis'}
FUNCTION F_GetCompany : WSTRING
VAR_INPUT
	
END_VAR

F_GetCompany := "Timberline Automation and Control Co.";

END_FUNCTION

// ---- Project Information/F_GetTitle.TcPOU
// This function has been automatically generated from the project information.
{attribute 'signature_flag' := '1073741824'}
{attribute 'TcGenerated'}
{attribute 'no-analysis'}
FUNCTION F_GetTitle : WSTRING
VAR_INPUT
	
END_VAR

F_GetTitle := "TAC_Events";

END_FUNCTION
